{attribute 'qualified_only'}
VAR_GLOBAL
	position: UINT := 0;
	velocity: UINT := 0;
	acceleration: UINT := 0;
	execute: BOOL := FALSE;
END_VAR

(* stored: Version 1.1.0.1, ProductVersion 3.1.4024.12
   GVL GVL_VARS1: Id {e45dfdf9-f4c5-4bdc-a76d-8754555a1000} *)
